				IF nSortBufferLogEnable.BUFFER_UPDATEDEST THEN
					sMessage := CONCAT('Item: ', TransportItemInSorter.ID);
					sMessage := CONCAT(sMessage,' Index: ');
					sMessage := CONCAT(sMessage, UDINT_TO_STRING(TransportSorterIndex));
					sMessage := CONCAT(sMessage,' New Dest: ');
					sMessage := CONCAT(sMessage, DINT_TO_STRING(TransportItemInSorter.Destination));
					sMessage := CONCAT(sMessage,' New Idx: ');
					sMessage := CONCAT(sMessage, DINT_TO_STRING(TransportItemInSorter.DestinationIdx));
					sMessage := CONCAT(sMessage,' New DeviceID ');
					sMessage := CONCAT(sMessage, TransportItemInSorter.DeviceID);
					// Write to the Error List
					ADSLOGSTR( msgCtrlMask := ADSLOG_MSGTYPE_HINT OR ADSLOG_MSGTYPE_LOG
						, msgFmtStr := CONCAT(st_Sorter.Config.Name, ' Dest Updated After Induct: %s')
						, strArg := sMessage);
				END_IF
			END_IF
			// Make sure that the destination update makes it to the item being inducted into the sorter
			IF st_UpdateItem.Item.ID <> '' THEN
				IF st_UpdateItem.Item.ID = TransportItemFound.ID THEN
					IF st_UpdateItem.Item.Destination <> TransportItemFound.Destination THEN
						IF nSortBufferLogEnable.BUFFER_UPDATEDEST THEN
							// Log the original destination
							sMessage := CONCAT('Item: ', st_UpdateItem.Item.ID);
							sMessage := CONCAT(sMessage, ' Pulses: ');
							sMessage := CONCAT(sMessage, UDINT_TO_STRING(st_Sorter.EncoderCounts));
							sMessage := CONCAT(sMessage,' Orig Dest: ');
							sMessage := CONCAT(sMessage, DINT_TO_STRING(st_UpdateItem.Item.Destination));
							sMessage := CONCAT(sMessage,' Orig Idx: ');
							sMessage := CONCAT(sMessage, DINT_TO_STRING(st_UpdateItem.Item.DestinationIdx));
							// Write to the Error List
							ADSLOGSTR( msgCtrlMask := ADSLOG_MSGTYPE_HINT OR ADSLOG_MSGTYPE_LOG
								, msgFmtStr := CONCAT(st_Sorter.Config.Name, ' Induct Dest Changed: %s')
								, strArg := sMessage);
						END_IF
						// Update the Destination and Index
						st_UpdateItem.Item.Destination := TransportItemFound.Destination;
						st_UpdateItem.Item.DestinationIdx := TransportItemFound.DestinationIdx;
						// Log the new destination
						IF nSortBufferLogEnable.BUFFER_UPDATEDEST THEN
							sMessage := CONCAT('Item: ', st_UpdateItem.Item.ID);
							sMessage := CONCAT(sMessage, ' Pulses: ');
							sMessage := CONCAT(sMessage, UDINT_TO_STRING(st_Sorter.EncoderCounts));
							sMessage := CONCAT(sMessage,' New Dest: ');
							sMessage := CONCAT(sMessage, DINT_TO_STRING(st_UpdateItem.Item.Destination));
							sMessage := CONCAT(sMessage,' New Idx: ');
							sMessage := CONCAT(sMessage, DINT_TO_STRING(st_UpdateItem.Item.DestinationIdx));
							// Write to the Error List
							ADSLOGSTR( msgCtrlMask := ADSLOG_MSGTYPE_HINT OR ADSLOG_MSGTYPE_LOG
								, msgFmtStr := CONCAT(st_Sorter.Config.Name, ' Induct Dest Changed: %s')
								, strArg := sMessage);
						END_IF
					END_IF
				END_IF
			ELSE
				IF nSortBufferLogEnable.BUFFER_UPDATEDEST THEN
					sMessage := CONCAT('Item: ', TransportItemInSorter.ID);
					sMessage := CONCAT(sMessage,' Index: ');
					sMessage := CONCAT(sMessage, UDINT_TO_STRING(TransportSorterIndex));
					sMessage := CONCAT(sMessage,' Orig Dest: ');
					sMessage := CONCAT(sMessage, DINT_TO_STRING(TransportItemInSorter.Destination));
					sMessage := CONCAT(sMessage,' Orig Idx: ');
					sMessage := CONCAT(sMessage, DINT_TO_STRING(TransportItemInSorter.DestinationIdx));
					// Write to the Error List
					ADSLOGSTR( msgCtrlMask := ADSLOG_MSGTYPE_HINT OR ADSLOG_MSGTYPE_LOG
						, msgFmtStr := CONCAT(st_Sorter.Config.Name, ' Dest Received After Induct: %s')
						, strArg := sMessage);
				END_IF
			END_IF
		END_IF
	END_IF

	// Put the updated record back into the array
	aItems[TransportSorterIndex] := TransportItemInSorter;
	
//==================================================
// 	Done procesing Transport information
//
//	Begin processing Update/Exit information
//==================================================
	
	// For exits, start from the current encoder count and work forward
	ExitSorterIndex := F_CalculateIndex(Offset := UpdateIndexCounter
										, InitialValue := st_Sorter.EncoderCounts
										, BufferSize := ItemsArraySize);

	// Identify the Item we are testing
	ExitItemInSorter := aItems[ExitSorterIndex];

	// Populated ID identifies an item in the sorter
	// Between the two Divert status codes indicates that the item has attempted to divert
	IF ExitItemInSorter.ID <> '' THEN
		// Capture the Item encoder index and the Item at the current index
		//  This represents the first item record for this item
		//  It is captured to log the start index to allow this first record to be updated
		//  when the item is completely diverted
		IF ExitItemFound.Item.ID = '' THEN
			ExitItemFound.Counts := ExitSorterIndex;
			ExitItemFound.Item := ExitItemInSorter;
			IF ExitItemFound.Item.Status = E_StatusCode.Divert_Complete THEN
				ExitComplete := TRUE;
			END_IF
		END_IF
		// When ExitComplete is TRUE, and the ID's match, clear out this Item
		IF ExitComplete THEN
			IF ExitItemInSorter.ID = ExitItemFound.Item.ID THEN
				IF aItems[ExitSorterIndex].ID <> '' THEN
					IF nSortBufferLogEnable.BUFFER_DUMP THEN
						sMessage := CONCAT('Item: ', aItems[ExitSorterIndex].ID);
						sMessage := CONCAT(sMessage,' Index: ');
						sMessage := CONCAT(sMessage, UDINT_TO_STRING(ExitSorterIndex));
						sMessage := CONCAT(sMessage,' Item Status: ');
						sMessage := CONCAT(sMessage, DINT_TO_STRING(aItems[ExitSorterIndex].Status));
						sMessage := CONCAT(sMessage,' Item Ext Status: ');
						sMessage := CONCAT(sMessage, DINT_TO_STRING(aItems[ExitSorterIndex].ExtStatus));
						// Write to the Error List
						ADSLOGSTR( msgCtrlMask := ADSLOG_MSGTYPE_HINT OR ADSLOG_MSGTYPE_LOG
							, msgFmtStr := CONCAT(st_Sorter.Config.Name, ' Exit Complete Dump Info: %s')
							, strArg := sMessage);
					END_IF
				END_IF
				aItems[ExitSorterIndex] := BlankItem;
			END_IF
		// When ExitComplete is FALSE, test for a diverting/diverted item
		ELSE
			// Detect when this item is in a diverting state
			IF (ExitItemInSorter.Status >= E_StatusCode.Diverting
			   OR ExitItemInSorter.Status <= E_StatusCode.Divert_Success)
			   THEN
			   	ExitInDivert := TRUE;
				(*
					Status value increase from Diverting to Divert_Complete
					Codes to indicate divert disposition are between Diverting and Divert_Detected
					Divert_Full and Diverting are set in FB_DivertDecision/FB_DivertControl
					Divert_Detected, Divert_Success, and Divert_Missed are set in FB_ConfirmCheck
				*)
				ExitDiverting := TRUE;
				IF ExitItemInSorter.Status = E_StatusCode.Divert_Detected THEN
					ExitDetected := TRUE;
				END_IF
				// Once the divert is successful, we are no longer "diverting"
				IF ExitItemInSorter.Status = E_StatusCode.Divert_Success THEN
					ExitSuccess := TRUE;
					ExitDiverting := FALSE;
				END_IF
				(*	
					ExitItemInSorter is the current item being examined
					ExitItemFound.Item is a copy of the Array item at ExitItemFound.Counts
					ExitItemFound.Counts references the Array index of the first record associated with this item
					When a Status/ExtStatus of greater value is detected, the first record Status/ExtStatus is overwritten
					The ExitItemFound.Item.Status/.ExtStatus is also updated
				*)
				IF ExitItemInSorter.Status > aItems[ExitItemFound.Counts].Status THEN
					aItems[ExitItemFound.Counts].Status := ExitItemInSorter.Status;
					ExitItemFound.Item.Status := ExitItemInSorter.Status;
				END_IF
				IF ExitItemInSorter.ExtStatus > aItems[ExitItemFound.Counts].ExtStatus THEN
					aItems[ExitItemFound.Counts].ExtStatus := ExitItemInSorter.ExtStatus;
					ExitItemFound.Item.ExtStatus := ExitItemInSorter.ExtStatus;
				END_IF
			END_IF
			aItems[ExitSorterIndex].Status := ExitItemFound.Item.Status;
		END_IF
	ELSE
		(*
			This path is followed when the ExitItemInSorter.ID is empty, which indicates
			that the array record associated with this index is not occupied

			ExitInDivert, ExitDiverting and ExitSuccess are all set while the .ID is not empty
		*)
		// This item was in a "diverting" state
		IF ExitInDivert THEN
			// This item is not currently diverting
			IF NOT ExitDiverting THEN
				// Only change to a Divert_Success if a Divert_Success was detected
				// Any other status is captured in the ELSE clause of the CASE statement
				IF ExitSuccess THEN
					ExitItemFound.Item.Status := E_StatusCode.Divert_Success;
				END_IF
				IF NOT (ExitItemFound.Item.DestinationIdx = Sorter.NUMBEROFDIVERTS)
				   OR (ExitItemFound.Item.DestinationIdx = Sorter.NUMBEROFDIVERTS AND aDiverts[ExitItemFound.Item.DestinationIdx].Config.IsDischarge)
				   THEN 
					ExitItemFound.Item.CapturedInMetrics := TRUE;
					ExitItemFound.Item.MessageType := E_MessageIds.TransportComplete_26;
					fb_UpdateBuffer.AddItem(ExitItemFound.Item);
					aItems[ExitItemFound.Counts].Status := E_StatusCode.Divert_Complete;
				END_IF
			END_IF
		END_IF
		// Clear the last detected Exit item
		ExitItemFound.Item := BlankItem;
		// Reset the Detection booleans
		ExitInDivert := FALSE;
		ExitDiverting := FALSE;
		ExitDetected := FALSE;
		ExitSuccess := FALSE;
		ExitComplete := FALSE;
	END_IF
END_FOR

// If the ID is populated, we didn't find a match to update
IF st_ToUpdate.Item.ID <> '' THEN
	IF nSortBufferLogEnable.BUFFER_UNASSIGNED THEN
		sMessage := CONCAT('Item: ', st_ToUpdate.Item.ID);
		// Write to the Error List
		ADSLOGSTR( msgCtrlMask := ADSLOG_MSGTYPE_HINT OR ADSLOG_MSGTYPE_LOG
			, msgFmtStr := CONCAT(st_Sorter.Config.Name, ' Item Not Updated: %s')
			, strArg := sMessage);
	END_IF
	st_ToUpdate.Item.Status := E_StatusCode.Assign_NotFound;
	st_ToUpdate.Item.DeviceID := st_Sorter.Config.Name;
	st_ToUpdate.Item.MessageType := E_MessageIds.TransportResponse_25;
	fb_UpDateBuffer.AddItem(st_ItemToAdd := st_ToUpdate.Item);
	st_ToUpdate.Item := BlankItem;
END_IF

END_PROGRAM

// ---- GlobalTextList.TcGTLO
TEXTLIST GlobalTextList
  645 = '%d'
  572 = '%s'
  787 = 'Captured'
  26 = 'Destination'
  290 = 'Device ID'
  976 = 'Diverter 1 Out'
  64 = 'Diverter 1 PE'
  977 = 'Diverter 2 Out'
  65 = 'Diverter 2 PE'
  978 = 'Diverter 3 Out'
  422 = 'Diverter 3 PE'
  979 = 'Diverter 4 Out'
  423 = 'Diverter 4 PE'
  980 = 'Diverter 5 Out'
  424 = 'Diverter 5 PE'
  950 = 'Encoder Counts'
  341 = 'Item ID (Barcode)'
  534 = 'Length'
  612 = 'Msg ID'
  425 = 'Sorter\n Barcode Read'
  426 = 'Sorter\nInduct PE'
  825 = 'Status'
  666 = 'Unique ID'
END_TEXTLIST

// ---- POUs/FunctionBlocks/Sorter/VISUs/SorterArray.TcVIS
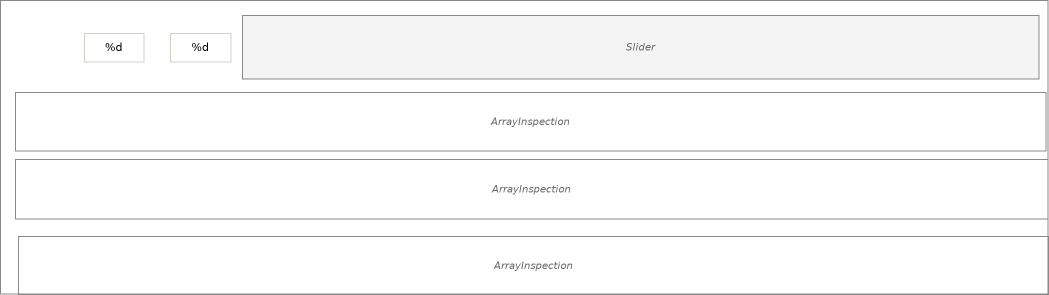
VISUALIZATION SorterArray  // 1049x295
    Frame (15,92 1031x59)
        shows ArrayInspection(st_ItemExt_Disp := MAIN.st_DisplayItem)
        shows ArrayInspection()
        shows ArrayInspection()
    Textfield (170,33 61x29), "%d", text variable: MAIN.nDisplayItemIndex
        OnMouseDown: write MAIN.nDisplayItemIndex via Edit
    Slider (242,15 797x64), variable: MAIN.nDisplayItemIndex, scale 0..100
    Textfield (84,33 60x29), "%d", text variable: MAIN.st_SorterEncoder.CurrentCount
    Frame (15,159 1033x60)
        shows ArrayInspection(st_ItemExt_Disp := ProcessBuffers_6040.st_DisplayItem)
    Frame (18,236 1031x59)
        shows ArrayInspection(st_ItemExt_Disp := SorterProgram.st_DisplayItem)
END_VISUALIZATION
